// Mitsubishi GX Developer project: PLC_PCO520L2   PLC: Q06UDEH

PROGRAM MANUAL
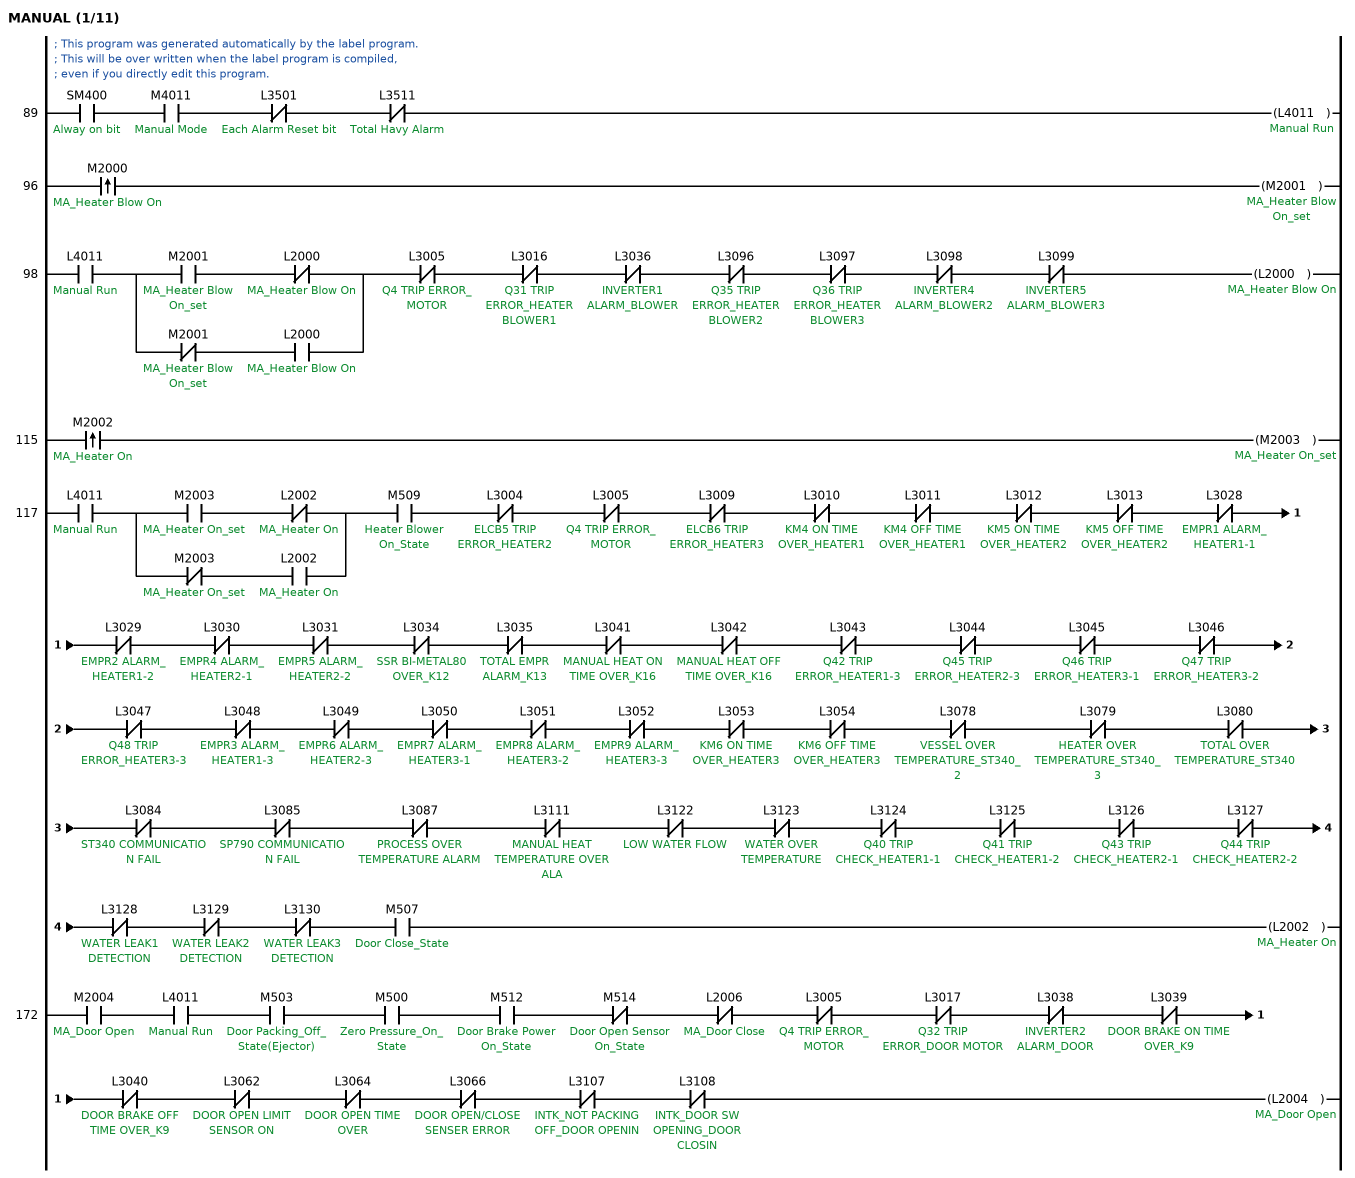
; This program was generated automatically by the label program.
; This will be over written when the label program is compiled,
; even if you directly edit this program.
89    LD      SM400  ; Alway on bit
      AND     M4011  ; Manual Mode
      ANI     L3501  ; Each Alarm Reset bit
      ANI     L3511  ; Total Havy Alarm
      OUT     L4011  ; Manual Run
; 
96    LDP     M2000  ; MA_Heater Blow On
      OUT     M2001  ; MA_Heater Blow On_set
98    LD      L4011  ; Manual Run
      LD      M2001  ; MA_Heater Blow On_set
      ANI     L2000  ; MA_Heater Blow On
      LDI     M2001  ; MA_Heater Blow On_set
      AND     L2000  ; MA_Heater Blow On
      ORB
      ANB
      ANI     L3005  ; Q4 TRIP ERROR_MOTOR
      ANI     L3016  ; Q31 TRIP ERROR_HEATER BLOWER1
      ANI     L3036  ; INVERTER1 ALARM_BLOWER
      ANI     L3096  ; Q35 TRIP ERROR_HEATER BLOWER2
      ANI     L3097  ; Q36 TRIP ERROR_HEATER BLOWER3
      ANI     L3098  ; INVERTER4 ALARM_BLOWER2
      ANI     L3099  ; INVERTER5 ALARM_BLOWER3
      OUT     L2000  ; MA_Heater Blow On
; 
115   LDP     M2002  ; MA_Heater On
      OUT     M2003  ; MA_Heater On_set
117   LD      L4011  ; Manual Run
      LD      M2003  ; MA_Heater On_set
      ANI     L2002  ; MA_Heater On
      LDI     M2003  ; MA_Heater On_set
      AND     L2002  ; MA_Heater On
      ORB
      ANB
      AND     M509  ; Heater Blower On_State
      ANI     L3004  ; ELCB5 TRIP ERROR_HEATER2
      ANI     L3005  ; Q4 TRIP ERROR_MOTOR
      ANI     L3009  ; ELCB6 TRIP ERROR_HEATER3
      ANI     L3010  ; KM4 ON TIME OVER_HEATER1
      ANI     L3011  ; KM4 OFF TIME OVER_HEATER1
      ANI     L3012  ; KM5 ON TIME OVER_HEATER2
      ANI     L3013  ; KM5 OFF TIME OVER_HEATER2
      ANI     L3028  ; EMPR1 ALARM_HEATER1-1
      ANI     L3029  ; EMPR2 ALARM_HEATER1-2
      ANI     L3030  ; EMPR4 ALARM_HEATER2-1
      ANI     L3031  ; EMPR5 ALARM_HEATER2-2
      ANI     L3034  ; SSR BI-METAL80 OVER_K12
      ANI     L3035  ; TOTAL EMPR ALARM_K13
      ANI     L3041  ; MANUAL HEAT ON TIME OVER_K16
      ANI     L3042  ; MANUAL HEAT OFF TIME OVER_K16
      ANI     L3043  ; Q42 TRIP ERROR_HEATER1-3
      ANI     L3044  ; Q45 TRIP ERROR_HEATER2-3
      ANI     L3045  ; Q46 TRIP ERROR_HEATER3-1
      ANI     L3046  ; Q47 TRIP ERROR_HEATER3-2
      ANI     L3047  ; Q48 TRIP ERROR_HEATER3-3
      ANI     L3048  ; EMPR3 ALARM_HEATER1-3
      ANI     L3049  ; EMPR6 ALARM_HEATER2-3
      ANI     L3050  ; EMPR7 ALARM_HEATER3-1
      ANI     L3051  ; EMPR8 ALARM_HEATER3-2
      ANI     L3052  ; EMPR9 ALARM_HEATER3-3
      ANI     L3053  ; KM6 ON TIME OVER_HEATER3
      ANI     L3054  ; KM6 OFF TIME OVER_HEATER3
      ANI     L3078  ; VESSEL OVER TEMPERATURE_ST340_2
      ANI     L3079  ; HEATER OVER TEMPERATURE_ST340_3
      ANI     L3080  ; TOTAL OVER TEMPERATURE_ST340
      ANI     L3084  ; ST340 COMMUNICATION FAIL
      ANI     L3085  ; SP790 COMMUNICATION FAIL
      ANI     L3087  ; PROCESS OVER TEMPERATURE ALARM
      ANI     L3111  ; MANUAL HEAT TEMPERATURE OVER ALA
      ANI     L3122  ; LOW WATER FLOW
      ANI     L3123  ; WATER OVER TEMPERATURE
      ANI     L3124  ; Q40 TRIP CHECK_HEATER1-1
      ANI     L3125  ; Q41 TRIP CHECK_HEATER1-2
      ANI     L3126  ; Q43 TRIP CHECK_HEATER2-1
      ANI     L3127  ; Q44 TRIP CHECK_HEATER2-2
      ANI     L3128  ; WATER LEAK1 DETECTION
      ANI     L3129  ; WATER LEAK2 DETECTION
      ANI     L3130  ; WATER LEAK3 DETECTION
      AND     M507  ; Door Close_State
      OUT     L2002  ; MA_Heater On
; 
172   LD      M2004  ; MA_Door Open
      AND     L4011  ; Manual Run
      AND     M503  ; Door Packing_Off_State(Ejector)
      AND     M500  ; Zero Pressure_On_State
      AND     M512  ; Door Brake Power On_State
      ANI     M514  ; Door Open Sensor On_State
      ANI     L2006  ; MA_Door Close
      ANI     L3005  ; Q4 TRIP ERROR_MOTOR
      ANI     L3017  ; Q32 TRIP ERROR_DOOR MOTOR
      ANI     L3038  ; INVERTER2 ALARM_DOOR
      ANI     L3039  ; DOOR BRAKE ON TIME OVER_K9
      ANI     L3040  ; DOOR BRAKE OFF TIME OVER_K9
      ANI     L3062  ; DOOR OPEN LIMIT SENSOR ON
      ANI     L3064  ; DOOR OPEN TIME OVER
      ANI     L3066  ; DOOR OPEN/CLOSE SENSER ERROR
      ANI     L3107  ; INTK_NOT PACKING OFF_DOOR OPENIN
      ANI     L3108  ; INTK_DOOR SW OPENING_DOOR CLOSIN
      OUT     L2004  ; MA_Door Open
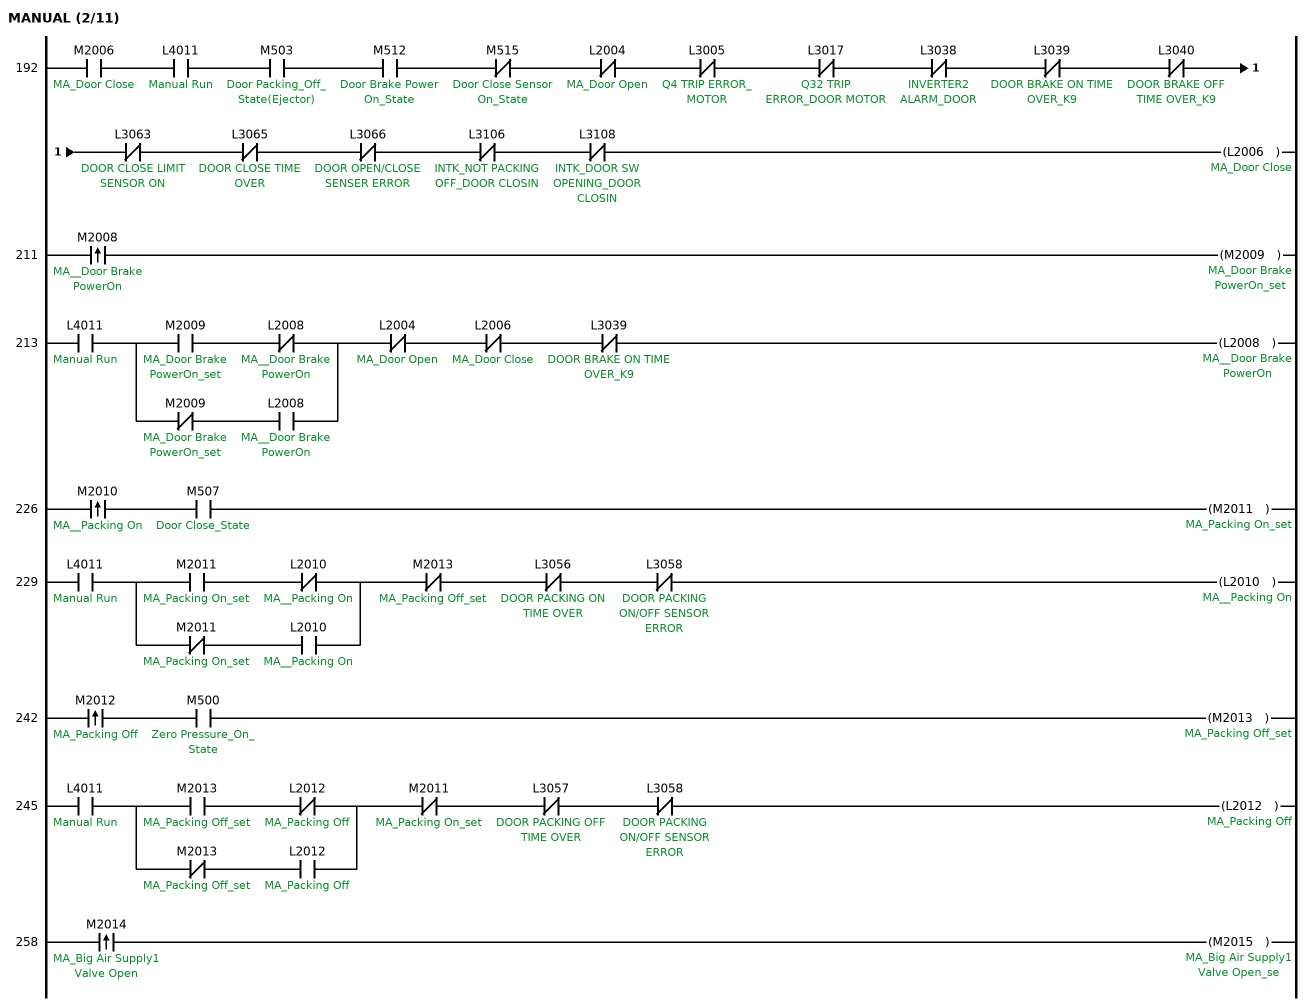
; 
192   LD      M2006  ; MA_Door Close
      AND     L4011  ; Manual Run
      AND     M503  ; Door Packing_Off_State(Ejector)
      AND     M512  ; Door Brake Power On_State
      ANI     M515  ; Door Close Sensor On_State
      ANI     L2004  ; MA_Door Open
      ANI     L3005  ; Q4 TRIP ERROR_MOTOR
      ANI     L3017  ; Q32 TRIP ERROR_DOOR MOTOR
      ANI     L3038  ; INVERTER2 ALARM_DOOR
      ANI     L3039  ; DOOR BRAKE ON TIME OVER_K9
      ANI     L3040  ; DOOR BRAKE OFF TIME OVER_K9
      ANI     L3063  ; DOOR CLOSE LIMIT SENSOR ON
      ANI     L3065  ; DOOR CLOSE TIME OVER
      ANI     L3066  ; DOOR OPEN/CLOSE SENSER ERROR
      ANI     L3106  ; INTK_NOT PACKING OFF_DOOR CLOSIN
      ANI     L3108  ; INTK_DOOR SW OPENING_DOOR CLOSIN
      OUT     L2006  ; MA_Door Close
; 
211   LDP     M2008  ; MA__Door Brake PowerOn
      OUT     M2009  ; MA_Door Brake PowerOn_set
213   LD      L4011  ; Manual Run
      LD      M2009  ; MA_Door Brake PowerOn_set
      ANI     L2008  ; MA__Door Brake PowerOn
      LDI     M2009  ; MA_Door Brake PowerOn_set
      AND     L2008  ; MA__Door Brake PowerOn
      ORB
      ANB
      ANI     L2004  ; MA_Door Open
      ANI     L2006  ; MA_Door Close
      ANI     L3039  ; DOOR BRAKE ON TIME OVER_K9
      OUT     L2008  ; MA__Door Brake PowerOn
; 
226   LDP     M2010  ; MA__Packing On
      AND     M507  ; Door Close_State
      OUT     M2011  ; MA_Packing On_set
229   LD      L4011  ; Manual Run
      LD      M2011  ; MA_Packing On_set
      ANI     L2010  ; MA__Packing On
      LDI     M2011  ; MA_Packing On_set
      AND     L2010  ; MA__Packing On
      ORB
      ANB
      ANI     M2013  ; MA_Packing Off_set
      ANI     L3056  ; DOOR PACKING ON TIME OVER
      ANI     L3058  ; DOOR PACKING ON/OFF SENSOR ERROR
      OUT     L2010  ; MA__Packing On
; 
242   LDP     M2012  ; MA_Packing Off
      AND     M500  ; Zero Pressure_On_State
      OUT     M2013  ; MA_Packing Off_set
245   LD      L4011  ; Manual Run
      LD      M2013  ; MA_Packing Off_set
      ANI     L2012  ; MA_Packing Off
      LDI     M2013  ; MA_Packing Off_set
      AND     L2012  ; MA_Packing Off
      ORB
      ANB
      ANI     M2011  ; MA_Packing On_set
      ANI     L3057  ; DOOR PACKING OFF TIME OVER
      ANI     L3058  ; DOOR PACKING ON/OFF SENSOR ERROR
      OUT     L2012  ; MA_Packing Off
; 
258   LDP     M2014  ; MA_Big Air Supply1 Valve Open
      OUT     M2015  ; MA_Big Air Supply1 Valve Open_se
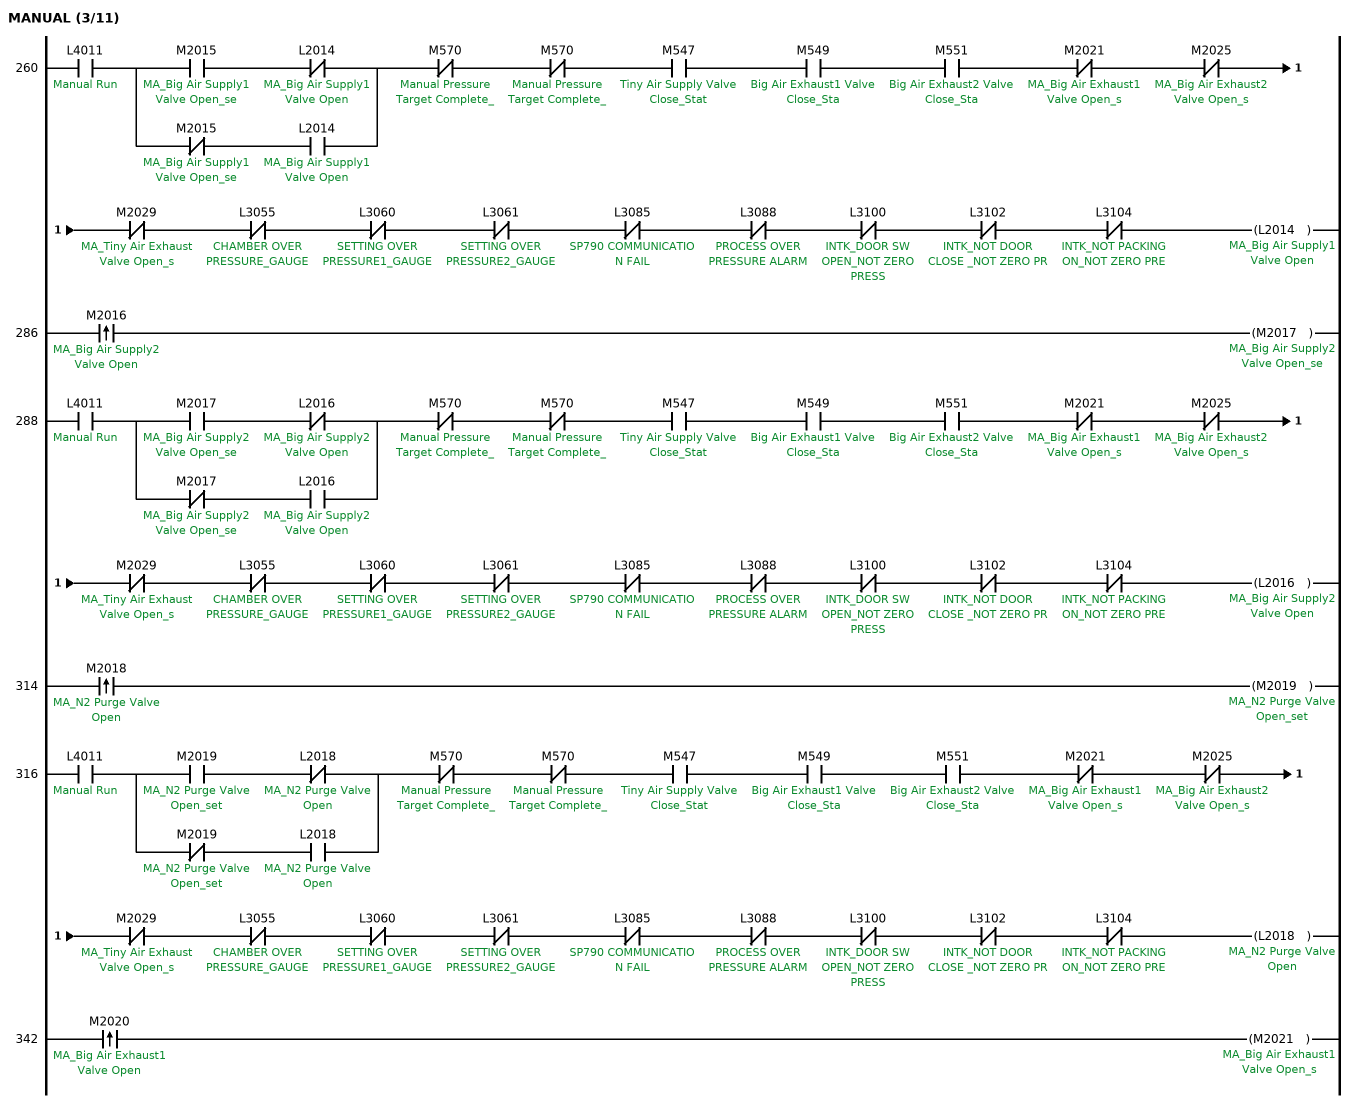
260   LD      L4011  ; Manual Run
      LD      M2015  ; MA_Big Air Supply1 Valve Open_se
      ANI     L2014  ; MA_Big Air Supply1 Valve Open
      LDI     M2015  ; MA_Big Air Supply1 Valve Open_se
      AND     L2014  ; MA_Big Air Supply1 Valve Open
      ORB
      ANB
      ANI     M570  ; Manual Pressure Target Complete_
      ANI     M570  ; Manual Pressure Target Complete_
      AND     M547  ; Tiny Air Supply Valve Close_Stat
      AND     M549  ; Big Air Exhaust1 Valve Close_Sta
      AND     M551  ; Big Air Exhaust2 Valve Close_Sta
      ANI     M2021  ; MA_Big Air Exhaust1 Valve Open_s
      ANI     M2025  ; MA_Big Air Exhaust2 Valve Open_s
      ANI     M2029  ; MA_Tiny Air Exhaust Valve Open_s
      ANI     L3055  ; CHAMBER OVER PRESSURE_GAUGE
      ANI     L3060  ; SETTING OVER PRESSURE1_GAUGE
      ANI     L3061  ; SETTING OVER PRESSURE2_GAUGE
      ANI     L3085  ; SP790 COMMUNICATION FAIL
      ANI     L3088  ; PROCESS OVER PRESSURE ALARM
      ANI     L3100  ; INTK_DOOR SW OPEN_NOT ZERO PRESS
      ANI     L3102  ; INTK_NOT DOOR CLOSE _NOT ZERO PR
      ANI     L3104  ; INTK_NOT PACKING ON_NOT ZERO PRE
      OUT     L2014  ; MA_Big Air Supply1 Valve Open
; 
286   LDP     M2016  ; MA_Big Air Supply2 Valve Open
      OUT     M2017  ; MA_Big Air Supply2 Valve Open_se
288   LD      L4011  ; Manual Run
      LD      M2017  ; MA_Big Air Supply2 Valve Open_se
      ANI     L2016  ; MA_Big Air Supply2 Valve Open
      LDI     M2017  ; MA_Big Air Supply2 Valve Open_se
      AND     L2016  ; MA_Big Air Supply2 Valve Open
      ORB
      ANB
      ANI     M570  ; Manual Pressure Target Complete_
      ANI     M570  ; Manual Pressure Target Complete_
      AND     M547  ; Tiny Air Supply Valve Close_Stat
      AND     M549  ; Big Air Exhaust1 Valve Close_Sta
      AND     M551  ; Big Air Exhaust2 Valve Close_Sta
      ANI     M2021  ; MA_Big Air Exhaust1 Valve Open_s
      ANI     M2025  ; MA_Big Air Exhaust2 Valve Open_s
      ANI     M2029  ; MA_Tiny Air Exhaust Valve Open_s
      ANI     L3055  ; CHAMBER OVER PRESSURE_GAUGE
      ANI     L3060  ; SETTING OVER PRESSURE1_GAUGE
      ANI     L3061  ; SETTING OVER PRESSURE2_GAUGE
      ANI     L3085  ; SP790 COMMUNICATION FAIL
      ANI     L3088  ; PROCESS OVER PRESSURE ALARM
      ANI     L3100  ; INTK_DOOR SW OPEN_NOT ZERO PRESS
      ANI     L3102  ; INTK_NOT DOOR CLOSE _NOT ZERO PR
      ANI     L3104  ; INTK_NOT PACKING ON_NOT ZERO PRE
      OUT     L2016  ; MA_Big Air Supply2 Valve Open
; 
314   LDP     M2018  ; MA_N2 Purge Valve Open
      OUT     M2019  ; MA_N2 Purge Valve Open_set
316   LD      L4011  ; Manual Run
      LD      M2019  ; MA_N2 Purge Valve Open_set
      ANI     L2018  ; MA_N2 Purge Valve Open
      LDI     M2019  ; MA_N2 Purge Valve Open_set
      AND     L2018  ; MA_N2 Purge Valve Open
      ORB
      ANB
      ANI     M570  ; Manual Pressure Target Complete_
      ANI     M570  ; Manual Pressure Target Complete_
      AND     M547  ; Tiny Air Supply Valve Close_Stat
      AND     M549  ; Big Air Exhaust1 Valve Close_Sta
      AND     M551  ; Big Air Exhaust2 Valve Close_Sta
      ANI     M2021  ; MA_Big Air Exhaust1 Valve Open_s
      ANI     M2025  ; MA_Big Air Exhaust2 Valve Open_s
      ANI     M2029  ; MA_Tiny Air Exhaust Valve Open_s
      ANI     L3055  ; CHAMBER OVER PRESSURE_GAUGE
      ANI     L3060  ; SETTING OVER PRESSURE1_GAUGE
      ANI     L3061  ; SETTING OVER PRESSURE2_GAUGE
      ANI     L3085  ; SP790 COMMUNICATION FAIL
      ANI     L3088  ; PROCESS OVER PRESSURE ALARM
      ANI     L3100  ; INTK_DOOR SW OPEN_NOT ZERO PRESS
      ANI     L3102  ; INTK_NOT DOOR CLOSE _NOT ZERO PR
      ANI     L3104  ; INTK_NOT PACKING ON_NOT ZERO PRE
      OUT     L2018  ; MA_N2 Purge Valve Open
; 
342   LDP     M2020  ; MA_Big Air Exhaust1 Valve Open
      OUT     M2021  ; MA_Big Air Exhaust1 Valve Open_s
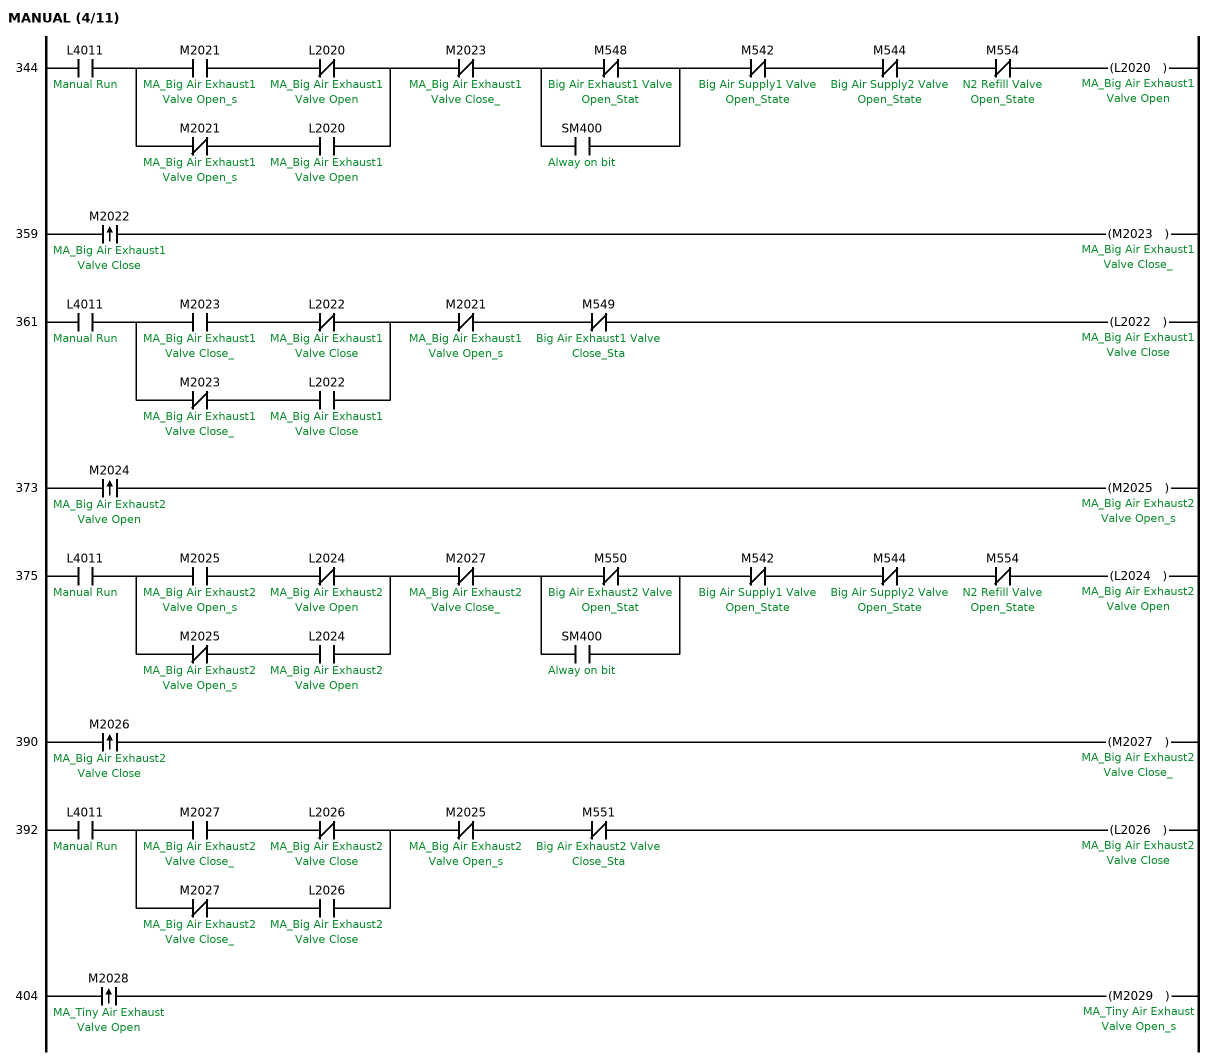
344   LD      L4011  ; Manual Run
      LD      M2021  ; MA_Big Air Exhaust1 Valve Open_s
      ANI     L2020  ; MA_Big Air Exhaust1 Valve Open
      LDI     M2021  ; MA_Big Air Exhaust1 Valve Open_s
      AND     L2020  ; MA_Big Air Exhaust1 Valve Open
      ORB
      ANB
      ANI     M2023  ; MA_Big Air Exhaust1 Valve Close_
      LDI     M548  ; Big Air Exhaust1 Valve Open_Stat
      OR      SM400  ; Alway on bit
      ANB
      ANI     M542  ; Big Air Supply1 Valve Open_State
      ANI     M544  ; Big Air Supply2 Valve Open_State
      ANI     M554  ; N2 Refill Valve Open_State
      OUT     L2020  ; MA_Big Air Exhaust1 Valve Open
359   LDP     M2022  ; MA_Big Air Exhaust1 Valve Close
      OUT     M2023  ; MA_Big Air Exhaust1 Valve Close_
361   LD      L4011  ; Manual Run
      LD      M2023  ; MA_Big Air Exhaust1 Valve Close_
      ANI     L2022  ; MA_Big Air Exhaust1 Valve Close
      LDI     M2023  ; MA_Big Air Exhaust1 Valve Close_
      AND     L2022  ; MA_Big Air Exhaust1 Valve Close
      ORB
      ANB
      ANI     M2021  ; MA_Big Air Exhaust1 Valve Open_s
      ANI     M549  ; Big Air Exhaust1 Valve Close_Sta
      OUT     L2022  ; MA_Big Air Exhaust1 Valve Close
; 
373   LDP     M2024  ; MA_Big Air Exhaust2 Valve Open
      OUT     M2025  ; MA_Big Air Exhaust2 Valve Open_s
375   LD      L4011  ; Manual Run
      LD      M2025  ; MA_Big Air Exhaust2 Valve Open_s
      ANI     L2024  ; MA_Big Air Exhaust2 Valve Open
      LDI     M2025  ; MA_Big Air Exhaust2 Valve Open_s
      AND     L2024  ; MA_Big Air Exhaust2 Valve Open
      ORB
      ANB
      ANI     M2027  ; MA_Big Air Exhaust2 Valve Close_
      LDI     M550  ; Big Air Exhaust2 Valve Open_Stat
      OR      SM400  ; Alway on bit
      ANB
      ANI     M542  ; Big Air Supply1 Valve Open_State
      ANI     M544  ; Big Air Supply2 Valve Open_State
      ANI     M554  ; N2 Refill Valve Open_State
      OUT     L2024  ; MA_Big Air Exhaust2 Valve Open
390   LDP     M2026  ; MA_Big Air Exhaust2 Valve Close
      OUT     M2027  ; MA_Big Air Exhaust2 Valve Close_
392   LD      L4011  ; Manual Run
      LD      M2027  ; MA_Big Air Exhaust2 Valve Close_
      ANI     L2026  ; MA_Big Air Exhaust2 Valve Close
      LDI     M2027  ; MA_Big Air Exhaust2 Valve Close_
      AND     L2026  ; MA_Big Air Exhaust2 Valve Close
      ORB
      ANB
      ANI     M2025  ; MA_Big Air Exhaust2 Valve Open_s
      ANI     M551  ; Big Air Exhaust2 Valve Close_Sta
      OUT     L2026  ; MA_Big Air Exhaust2 Valve Close
; 
404   LDP     M2028  ; MA_Tiny Air Exhaust Valve Open
      OUT     M2029  ; MA_Tiny Air Exhaust Valve Open_s
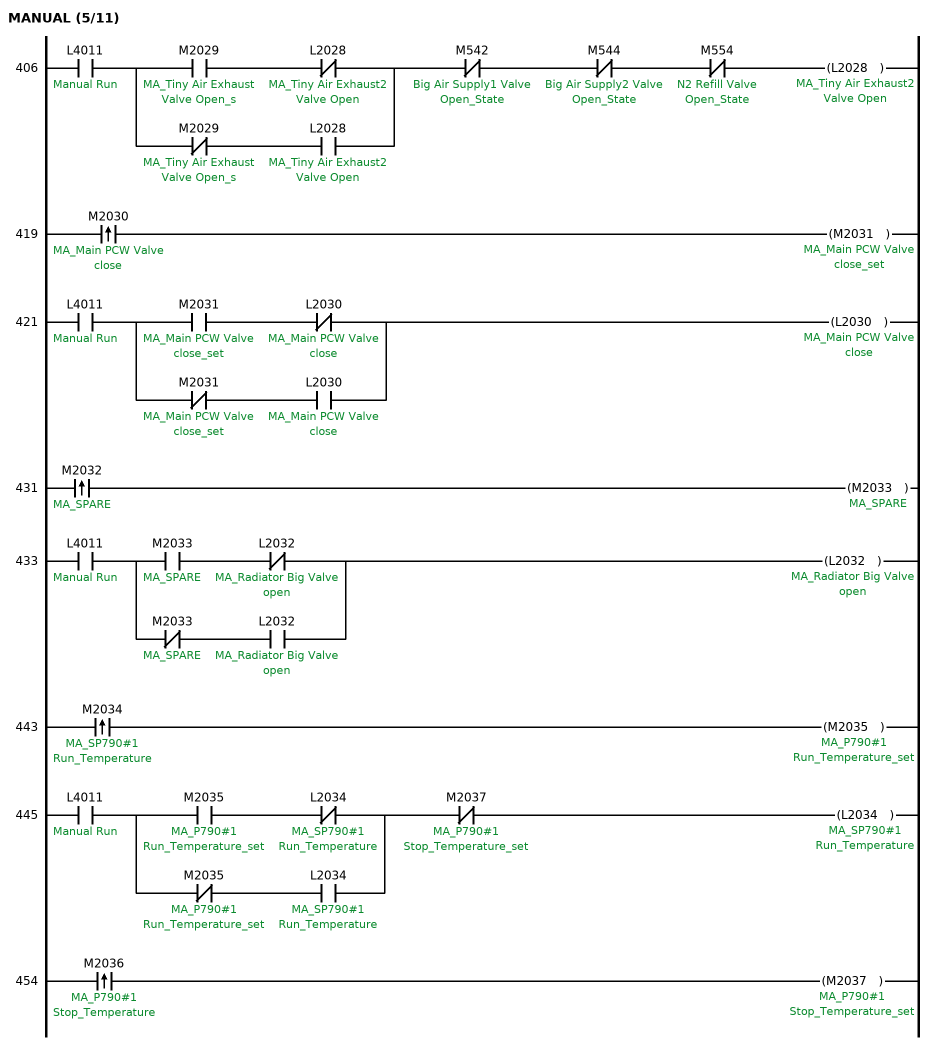
406   LD      L4011  ; Manual Run
      LD      M2029  ; MA_Tiny Air Exhaust Valve Open_s
      ANI     L2028  ; MA_Tiny Air Exhaust2 Valve Open
      LDI     M2029  ; MA_Tiny Air Exhaust Valve Open_s
      AND     L2028  ; MA_Tiny Air Exhaust2 Valve Open
      ORB
      ANB
      ANI     M542  ; Big Air Supply1 Valve Open_State
      ANI     M544  ; Big Air Supply2 Valve Open_State
      ANI     M554  ; N2 Refill Valve Open_State
      OUT     L2028  ; MA_Tiny Air Exhaust2 Valve Open
; 
419   LDP     M2030  ; MA_Main PCW Valve close
      OUT     M2031  ; MA_Main PCW Valve close_set
421   LD      L4011  ; Manual Run
      LD      M2031  ; MA_Main PCW Valve close_set
      ANI     L2030  ; MA_Main PCW Valve close
      LDI     M2031  ; MA_Main PCW Valve close_set
      AND     L2030  ; MA_Main PCW Valve close
      ORB
      ANB
      OUT     L2030  ; MA_Main PCW Valve close
; 
431   LDP     M2032  ; MA_SPARE
      OUT     M2033  ; MA_SPARE
433   LD      L4011  ; Manual Run
      LD      M2033  ; MA_SPARE
      ANI     L2032  ; MA_Radiator Big Valve open
      LDI     M2033  ; MA_SPARE
      AND     L2032  ; MA_Radiator Big Valve open
      ORB
      ANB
      OUT     L2032  ; MA_Radiator Big Valve open
; 
443   LDP     M2034  ; MA_SP790#1 Run_Temperature
      OUT     M2035  ; MA_P790#1 Run_Temperature_set
445   LD      L4011  ; Manual Run
      LD      M2035  ; MA_P790#1 Run_Temperature_set
      ANI     L2034  ; MA_SP790#1 Run_Temperature
      LDI     M2035  ; MA_P790#1 Run_Temperature_set
      AND     L2034  ; MA_SP790#1 Run_Temperature
      ORB
      ANB
      ANI     M2037  ; MA_P790#1 Stop_Temperature_set
      OUT     L2034  ; MA_SP790#1 Run_Temperature
454   LDP     M2036  ; MA_P790#1 Stop_Temperature
      OUT     M2037  ; MA_P790#1 Stop_Temperature_set
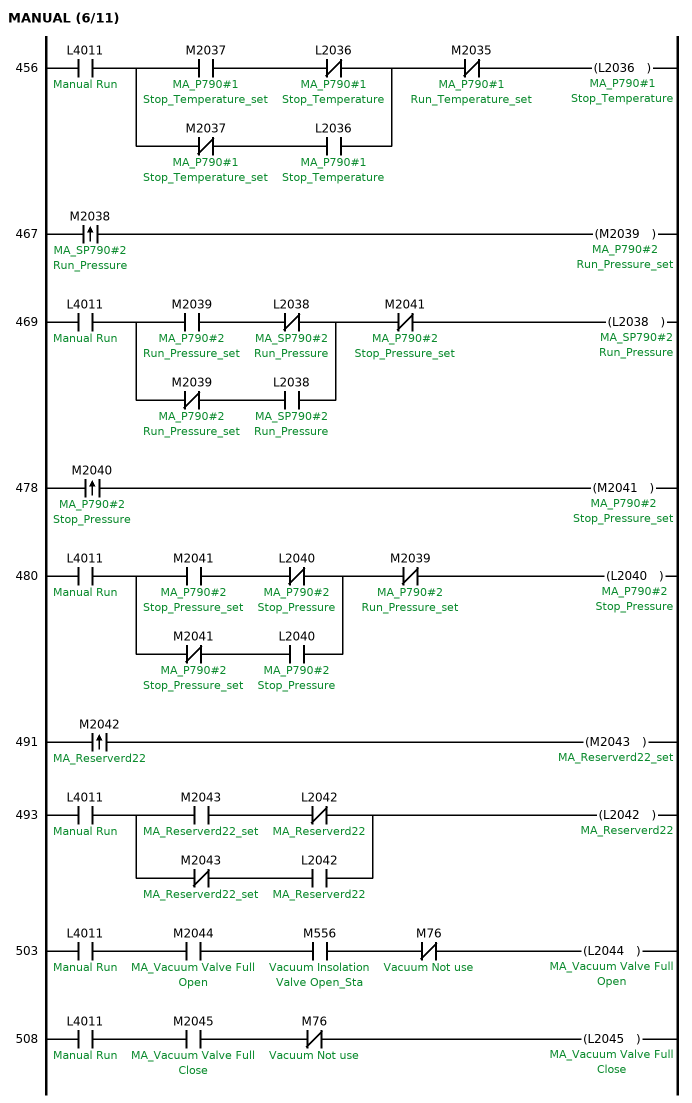
456   LD      L4011  ; Manual Run
      LD      M2037  ; MA_P790#1 Stop_Temperature_set
      ANI     L2036  ; MA_P790#1 Stop_Temperature
      LDI     M2037  ; MA_P790#1 Stop_Temperature_set
      AND     L2036  ; MA_P790#1 Stop_Temperature
      ORB
      ANB
      ANI     M2035  ; MA_P790#1 Run_Temperature_set
      OUT     L2036  ; MA_P790#1 Stop_Temperature
; 
467   LDP     M2038  ; MA_SP790#2 Run_Pressure
      OUT     M2039  ; MA_P790#2 Run_Pressure_set
469   LD      L4011  ; Manual Run
      LD      M2039  ; MA_P790#2 Run_Pressure_set
      ANI     L2038  ; MA_SP790#2 Run_Pressure
      LDI     M2039  ; MA_P790#2 Run_Pressure_set
      AND     L2038  ; MA_SP790#2 Run_Pressure
      ORB
      ANB
      ANI     M2041  ; MA_P790#2 Stop_Pressure_set
      OUT     L2038  ; MA_SP790#2 Run_Pressure
478   LDP     M2040  ; MA_P790#2 Stop_Pressure
      OUT     M2041  ; MA_P790#2 Stop_Pressure_set
480   LD      L4011  ; Manual Run
      LD      M2041  ; MA_P790#2 Stop_Pressure_set
      ANI     L2040  ; MA_P790#2 Stop_Pressure
      LDI     M2041  ; MA_P790#2 Stop_Pressure_set
      AND     L2040  ; MA_P790#2 Stop_Pressure
      ORB
      ANB
      ANI     M2039  ; MA_P790#2 Run_Pressure_set
      OUT     L2040  ; MA_P790#2 Stop_Pressure
; 
491   LDP     M2042  ; MA_Reserverd22
      OUT     M2043  ; MA_Reserverd22_set
493   LD      L4011  ; Manual Run
      LD      M2043  ; MA_Reserverd22_set
      ANI     L2042  ; MA_Reserverd22
      LDI     M2043  ; MA_Reserverd22_set
      AND     L2042  ; MA_Reserverd22
      ORB
      ANB
      OUT     L2042  ; MA_Reserverd22
; 
503   LD      L4011  ; Manual Run
      AND     M2044  ; MA_Vacuum Valve Full Open
      AND     M556  ; Vacuum Insolation Valve Open_Sta
      ANI     M76  ; Vacuum Not use
      OUT     L2044  ; MA_Vacuum Valve Full Open
508   LD      L4011  ; Manual Run
      AND     M2045  ; MA_Vacuum Valve Full Close
      ANI     M76  ; Vacuum Not use
      OUT     L2045  ; MA_Vacuum Valve Full Close
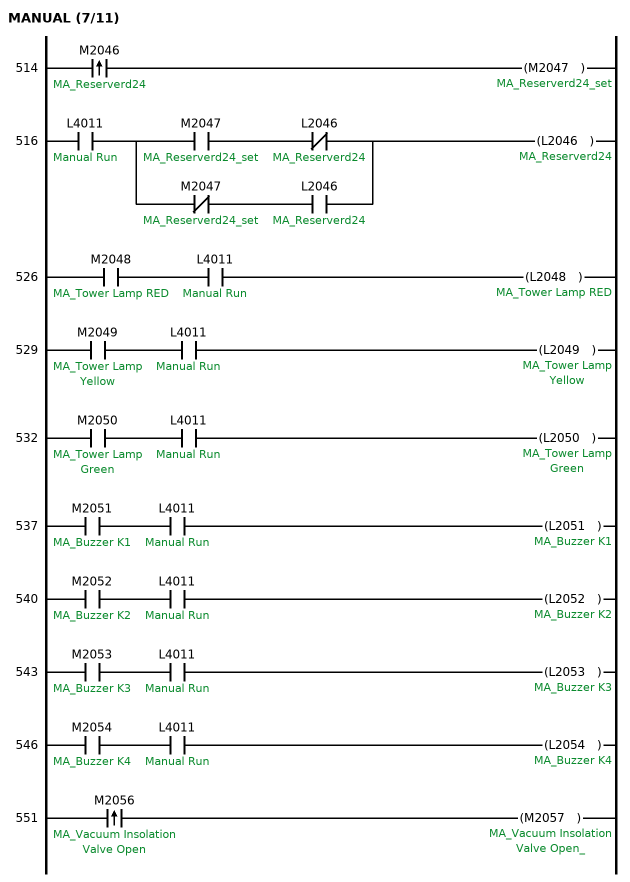
; 
514   LDP     M2046  ; MA_Reserverd24
      OUT     M2047  ; MA_Reserverd24_set
516   LD      L4011  ; Manual Run
      LD      M2047  ; MA_Reserverd24_set
      ANI     L2046  ; MA_Reserverd24
      LDI     M2047  ; MA_Reserverd24_set
      AND     L2046  ; MA_Reserverd24
      ORB
      ANB
      OUT     L2046  ; MA_Reserverd24
; 
526   LD      M2048  ; MA_Tower Lamp RED
      AND     L4011  ; Manual Run
      OUT     L2048  ; MA_Tower Lamp RED
529   LD      M2049  ; MA_Tower Lamp Yellow
      AND     L4011  ; Manual Run
      OUT     L2049  ; MA_Tower Lamp Yellow
532   LD      M2050  ; MA_Tower Lamp Green
      AND     L4011  ; Manual Run
      OUT     L2050  ; MA_Tower Lamp Green
; 
537   LD      M2051  ; MA_Buzzer K1
      AND     L4011  ; Manual Run
      OUT     L2051  ; MA_Buzzer K1
540   LD      M2052  ; MA_Buzzer K2
      AND     L4011  ; Manual Run
      OUT     L2052  ; MA_Buzzer K2
543   LD      M2053  ; MA_Buzzer K3
      AND     L4011  ; Manual Run
      OUT     L2053  ; MA_Buzzer K3
546   LD      M2054  ; MA_Buzzer K4
      AND     L4011  ; Manual Run
      OUT     L2054  ; MA_Buzzer K4
; 
551   LDP     M2056  ; MA_Vacuum Insolation Valve Open
      OUT     M2057  ; MA_Vacuum Insolation Valve Open_
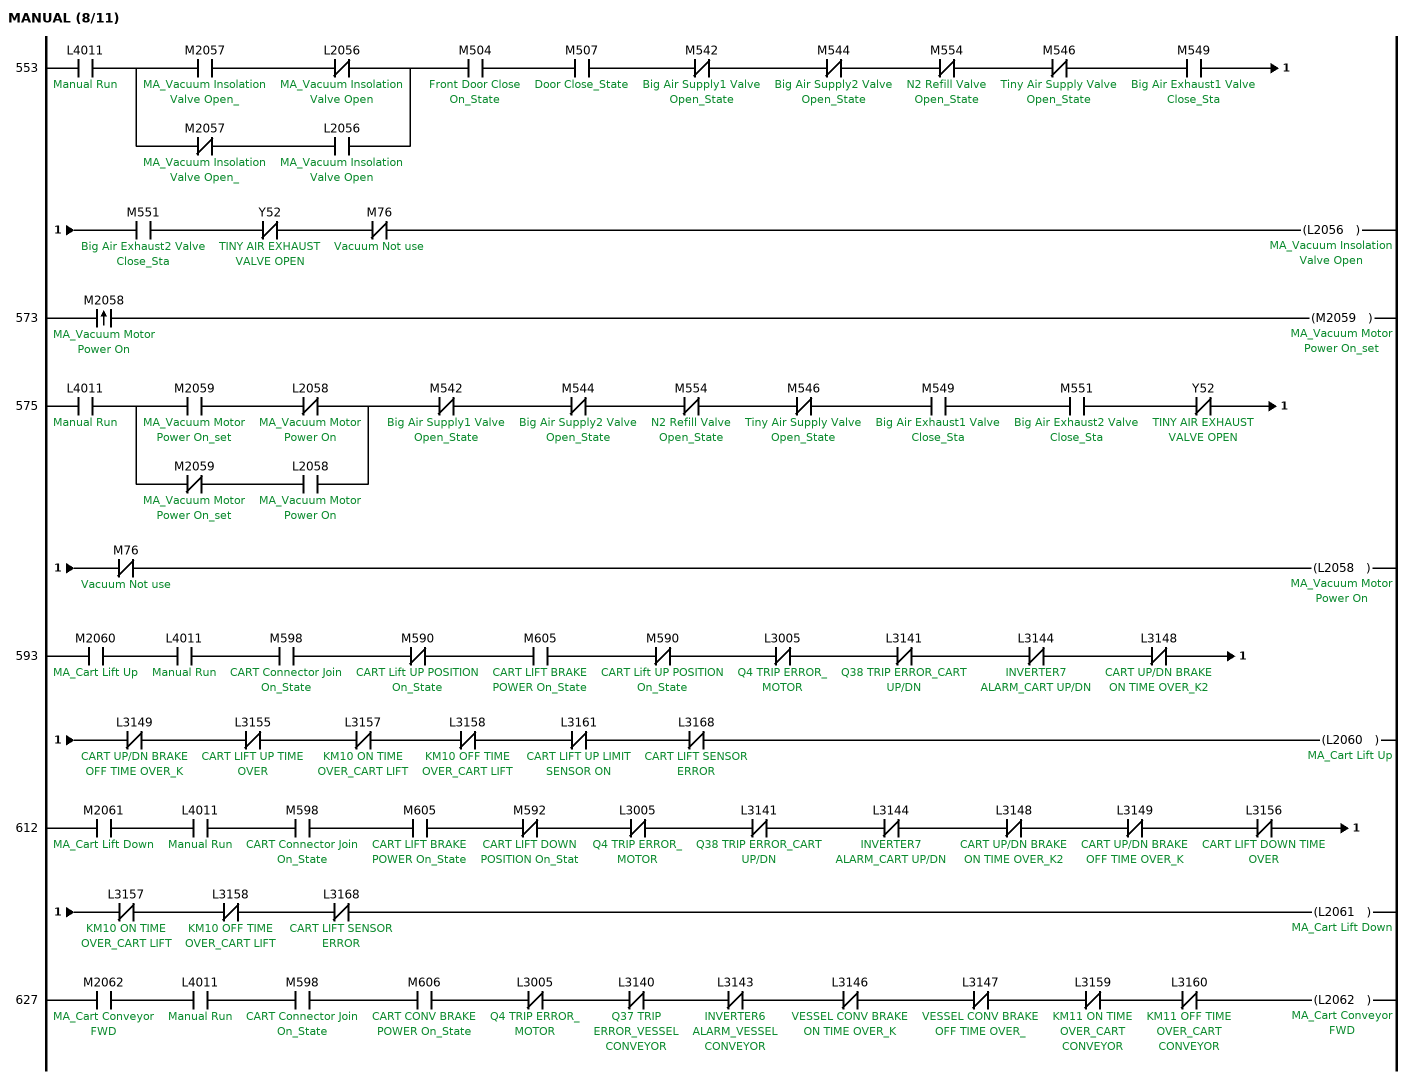
553   LD      L4011  ; Manual Run
      LD      M2057  ; MA_Vacuum Insolation Valve Open_
      ANI     L2056  ; MA_Vacuum Insolation Valve Open
      LDI     M2057  ; MA_Vacuum Insolation Valve Open_
      AND     L2056  ; MA_Vacuum Insolation Valve Open
      ORB
      ANB
      AND     M504  ; Front Door Close On_State
      AND     M507  ; Door Close_State
      ANI     M542  ; Big Air Supply1 Valve Open_State
      ANI     M544  ; Big Air Supply2 Valve Open_State
      ANI     M554  ; N2 Refill Valve Open_State
      ANI     M546  ; Tiny Air Supply Valve Open_State
      AND     M549  ; Big Air Exhaust1 Valve Close_Sta
      AND     M551  ; Big Air Exhaust2 Valve Close_Sta
      ANI     Y52  ; TINY AIR EXHAUST VALVE OPEN
      ANI     M76  ; Vacuum Not use
      OUT     L2056  ; MA_Vacuum Insolation Valve Open
; 
573   LDP     M2058  ; MA_Vacuum Motor Power On
      OUT     M2059  ; MA_Vacuum Motor Power On_set
575   LD      L4011  ; Manual Run
      LD      M2059  ; MA_Vacuum Motor Power On_set
      ANI     L2058  ; MA_Vacuum Motor Power On
      LDI     M2059  ; MA_Vacuum Motor Power On_set
      AND     L2058  ; MA_Vacuum Motor Power On
      ORB
      ANB
      ANI     M542  ; Big Air Supply1 Valve Open_State
      ANI     M544  ; Big Air Supply2 Valve Open_State
      ANI     M554  ; N2 Refill Valve Open_State
      ANI     M546  ; Tiny Air Supply Valve Open_State
      AND     M549  ; Big Air Exhaust1 Valve Close_Sta
      AND     M551  ; Big Air Exhaust2 Valve Close_Sta
      ANI     Y52  ; TINY AIR EXHAUST VALVE OPEN
      ANI     M76  ; Vacuum Not use
      OUT     L2058  ; MA_Vacuum Motor Power On
; 
593   LD      M2060  ; MA_Cart Lift Up
      AND     L4011  ; Manual Run
      AND     M598  ; CART Connector Join On_State
      ANI     M590  ; CART Lift UP POSITION On_State
      AND     M605  ; CART LIFT BRAKE POWER On_State
      ANI     M590  ; CART Lift UP POSITION On_State
      ANI     L3005  ; Q4 TRIP ERROR_MOTOR
      ANI     L3141  ; Q38 TRIP ERROR_CART UP/DN
      ANI     L3144  ; INVERTER7 ALARM_CART UP/DN
      ANI     L3148  ; CART UP/DN BRAKE ON TIME OVER_K2
      ANI     L3149  ; CART UP/DN BRAKE OFF TIME OVER_K
      ANI     L3155  ; CART LIFT UP TIME OVER
      ANI     L3157  ; KM10 ON TIME OVER_CART LIFT
      ANI     L3158  ; KM10 OFF TIME OVER_CART LIFT
      ANI     L3161  ; CART LIFT UP LIMIT SENSOR ON
      ANI     L3168  ; CART LIFT SENSOR ERROR
      OUT     L2060  ; MA_Cart Lift Up
; 
612   LD      M2061  ; MA_Cart Lift Down
      AND     L4011  ; Manual Run
      AND     M598  ; CART Connector Join On_State
      AND     M605  ; CART LIFT BRAKE POWER On_State
      ANI     M592  ; CART LIFT DOWN  POSITION On_Stat
      ANI     L3005  ; Q4 TRIP ERROR_MOTOR
      ANI     L3141  ; Q38 TRIP ERROR_CART UP/DN
      ANI     L3144  ; INVERTER7 ALARM_CART UP/DN
      ANI     L3148  ; CART UP/DN BRAKE ON TIME OVER_K2
      ANI     L3149  ; CART UP/DN BRAKE OFF TIME OVER_K
      ANI     L3156  ; CART LIFT DOWN TIME OVER
      ANI     L3157  ; KM10 ON TIME OVER_CART LIFT
      ANI     L3158  ; KM10 OFF TIME OVER_CART LIFT
      ANI     L3168  ; CART LIFT SENSOR ERROR
      OUT     L2061  ; MA_Cart Lift Down
627   LD      M2062  ; MA_Cart Conveyor FWD
      AND     L4011  ; Manual Run
      AND     M598  ; CART Connector Join On_State
      AND     M606  ; CART CONV BRAKE POWER On_State
      ANI     L3005  ; Q4 TRIP ERROR_MOTOR
      ANI     L3140  ; Q37 TRIP ERROR_VESSEL CONVEYOR
      ANI     L3143  ; INVERTER6 ALARM_VESSEL CONVEYOR
      ANI     L3146  ; VESSEL CONV BRAKE ON TIME OVER_K
      ANI     L3147  ; VESSEL CONV BRAKE OFF TIME OVER_
      ANI     L3159  ; KM11 ON TIME OVER_CART CONVEYOR
      ANI     L3160  ; KM11 OFF TIME OVER_CART CONVEYOR
      OUT     L2062  ; MA_Cart Conveyor FWD
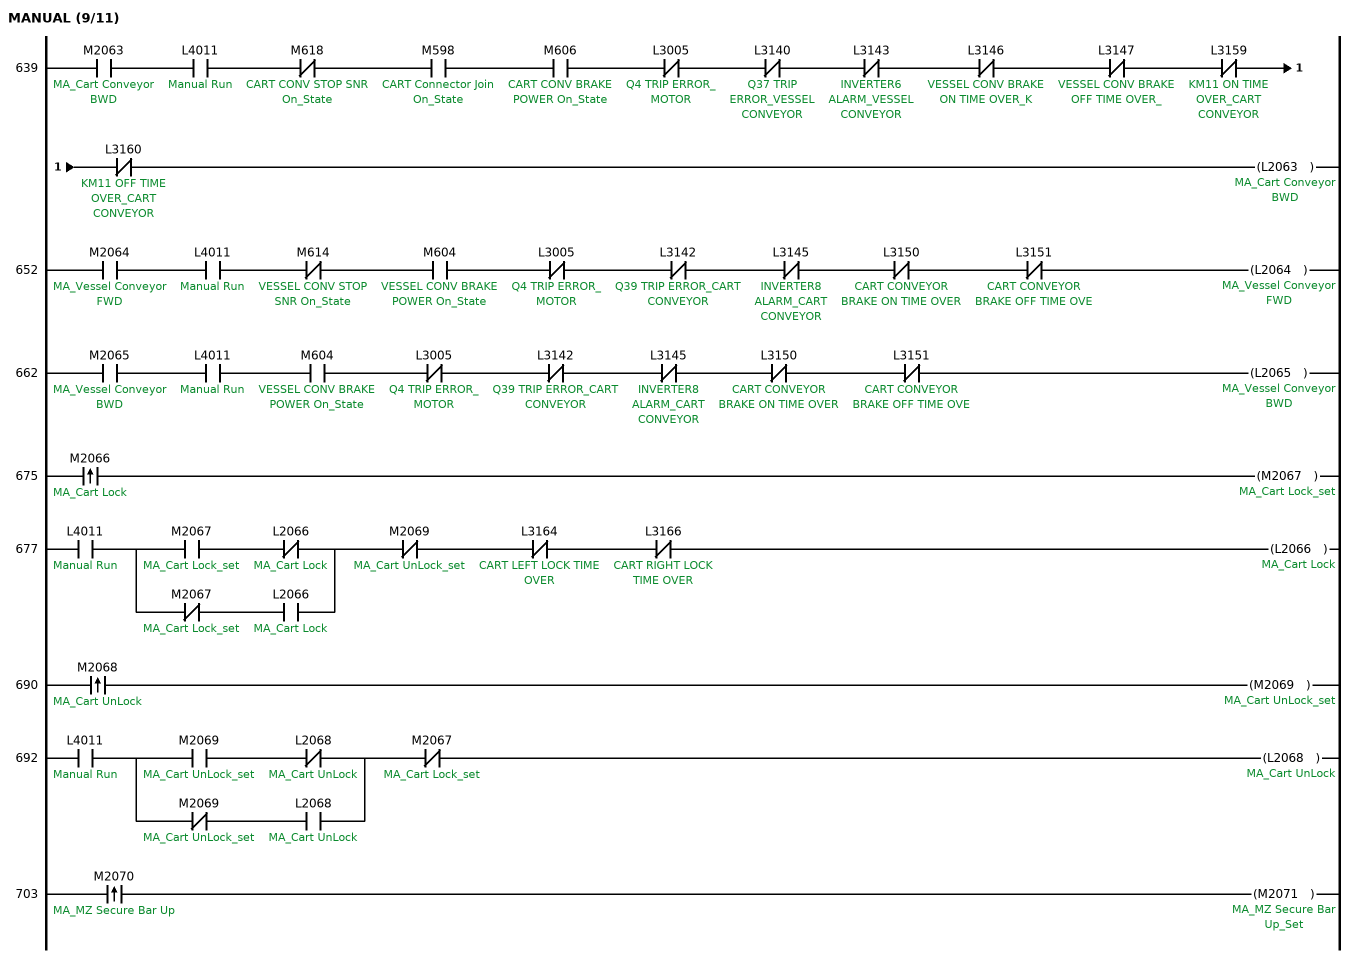
639   LD      M2063  ; MA_Cart Conveyor BWD
      AND     L4011  ; Manual Run
      ANI     M618  ; CART CONV STOP SNR On_State
      AND     M598  ; CART Connector Join On_State
      AND     M606  ; CART CONV BRAKE POWER On_State
      ANI     L3005  ; Q4 TRIP ERROR_MOTOR
      ANI     L3140  ; Q37 TRIP ERROR_VESSEL CONVEYOR
      ANI     L3143  ; INVERTER6 ALARM_VESSEL CONVEYOR
      ANI     L3146  ; VESSEL CONV BRAKE ON TIME OVER_K
      ANI     L3147  ; VESSEL CONV BRAKE OFF TIME OVER_
      ANI     L3159  ; KM11 ON TIME OVER_CART CONVEYOR
      ANI     L3160  ; KM11 OFF TIME OVER_CART CONVEYOR
      OUT     L2063  ; MA_Cart Conveyor BWD
652   LD      M2064  ; MA_Vessel Conveyor FWD
      AND     L4011  ; Manual Run
      ANI     M614  ; VESSEL CONV STOP SNR On_State
      AND     M604  ; VESSEL CONV BRAKE POWER On_State
      ANI     L3005  ; Q4 TRIP ERROR_MOTOR
      ANI     L3142  ; Q39 TRIP ERROR_CART CONVEYOR
      ANI     L3145  ; INVERTER8 ALARM_CART CONVEYOR
      ANI     L3150  ; CART CONVEYOR BRAKE ON TIME OVER
      ANI     L3151  ; CART CONVEYOR BRAKE OFF TIME OVE
      OUT     L2064  ; MA_Vessel Conveyor FWD
662   LD      M2065  ; MA_Vessel Conveyor BWD
      AND     L4011  ; Manual Run
      AND     M604  ; VESSEL CONV BRAKE POWER On_State
      ANI     L3005  ; Q4 TRIP ERROR_MOTOR
      ANI     L3142  ; Q39 TRIP ERROR_CART CONVEYOR
      ANI     L3145  ; INVERTER8 ALARM_CART CONVEYOR
      ANI     L3150  ; CART CONVEYOR BRAKE ON TIME OVER
      ANI     L3151  ; CART CONVEYOR BRAKE OFF TIME OVE
      OUT     L2065  ; MA_Vessel Conveyor BWD
; 
; 
675   LDP     M2066  ; MA_Cart Lock
      OUT     M2067  ; MA_Cart Lock_set
677   LD      L4011  ; Manual Run
      LD      M2067  ; MA_Cart Lock_set
      ANI     L2066  ; MA_Cart Lock
      LDI     M2067  ; MA_Cart Lock_set
      AND     L2066  ; MA_Cart Lock
      ORB
      ANB
      ANI     M2069  ; MA_Cart UnLock_set
      ANI     L3164  ; CART LEFT LOCK TIME OVER
      ANI     L3166  ; CART RIGHT LOCK TIME OVER
      OUT     L2066  ; MA_Cart Lock
; 
690   LDP     M2068  ; MA_Cart UnLock
      OUT     M2069  ; MA_Cart UnLock_set
692   LD      L4011  ; Manual Run
      LD      M2069  ; MA_Cart UnLock_set
      ANI     L2068  ; MA_Cart UnLock
      LDI     M2069  ; MA_Cart UnLock_set
      AND     L2068  ; MA_Cart UnLock
      ORB
      ANB
      ANI     M2067  ; MA_Cart Lock_set
      OUT     L2068  ; MA_Cart UnLock
; 
703   LDP     M2070  ; MA_MZ Secure Bar Up
      OUT     M2071  ; MA_MZ Secure Bar Up_Set
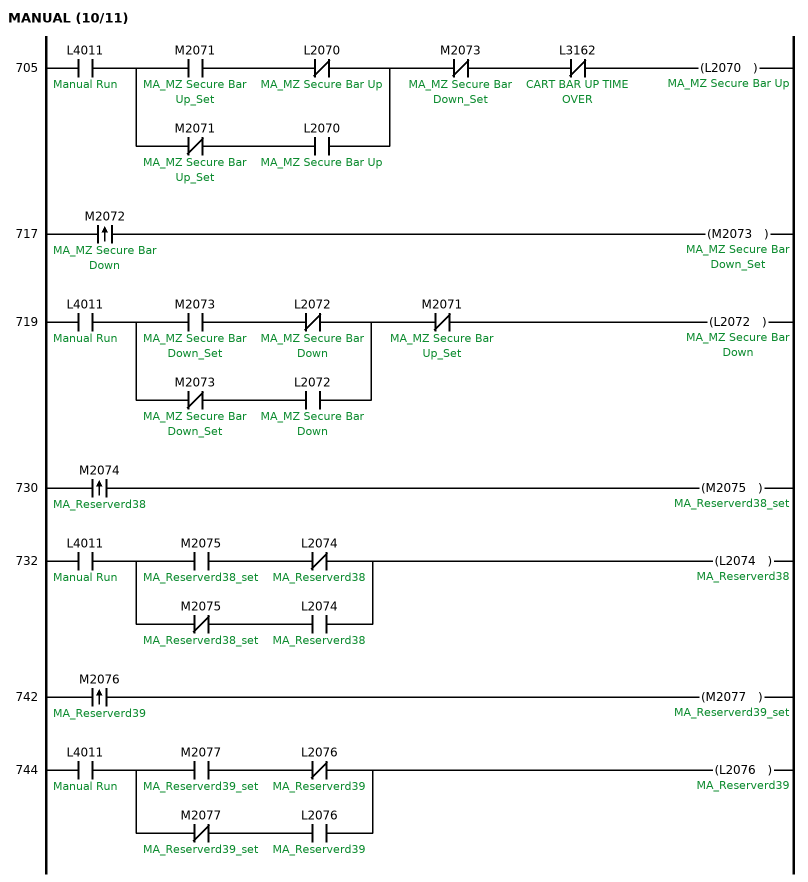
705   LD      L4011  ; Manual Run
      LD      M2071  ; MA_MZ Secure Bar Up_Set
      ANI     L2070  ; MA_MZ Secure Bar Up
      LDI     M2071  ; MA_MZ Secure Bar Up_Set
      AND     L2070  ; MA_MZ Secure Bar Up
      ORB
      ANB
      ANI     M2073  ; MA_MZ Secure Bar Down_Set
      ANI     L3162  ; CART BAR UP TIME OVER
      OUT     L2070  ; MA_MZ Secure Bar Up
; 
717   LDP     M2072  ; MA_MZ Secure Bar Down
      OUT     M2073  ; MA_MZ Secure Bar Down_Set
719   LD      L4011  ; Manual Run
      LD      M2073  ; MA_MZ Secure Bar Down_Set
      ANI     L2072  ; MA_MZ Secure Bar Down
      LDI     M2073  ; MA_MZ Secure Bar Down_Set
      AND     L2072  ; MA_MZ Secure Bar Down
      ORB
      ANB
      ANI     M2071  ; MA_MZ Secure Bar Up_Set
      OUT     L2072  ; MA_MZ Secure Bar Down
; 
730   LDP     M2074  ; MA_Reserverd38
      OUT     M2075  ; MA_Reserverd38_set
732   LD      L4011  ; Manual Run
      LD      M2075  ; MA_Reserverd38_set
      ANI     L2074  ; MA_Reserverd38
      LDI     M2075  ; MA_Reserverd38_set
      AND     L2074  ; MA_Reserverd38
      ORB
      ANB
      OUT     L2074  ; MA_Reserverd38
; 
742   LDP     M2076  ; MA_Reserverd39
      OUT     M2077  ; MA_Reserverd39_set
744   LD      L4011  ; Manual Run
      LD      M2077  ; MA_Reserverd39_set
      ANI     L2076  ; MA_Reserverd39
      LDI     M2077  ; MA_Reserverd39_set
      AND     L2076  ; MA_Reserverd39
      ORB
      ANB
      OUT     L2076  ; MA_Reserverd39
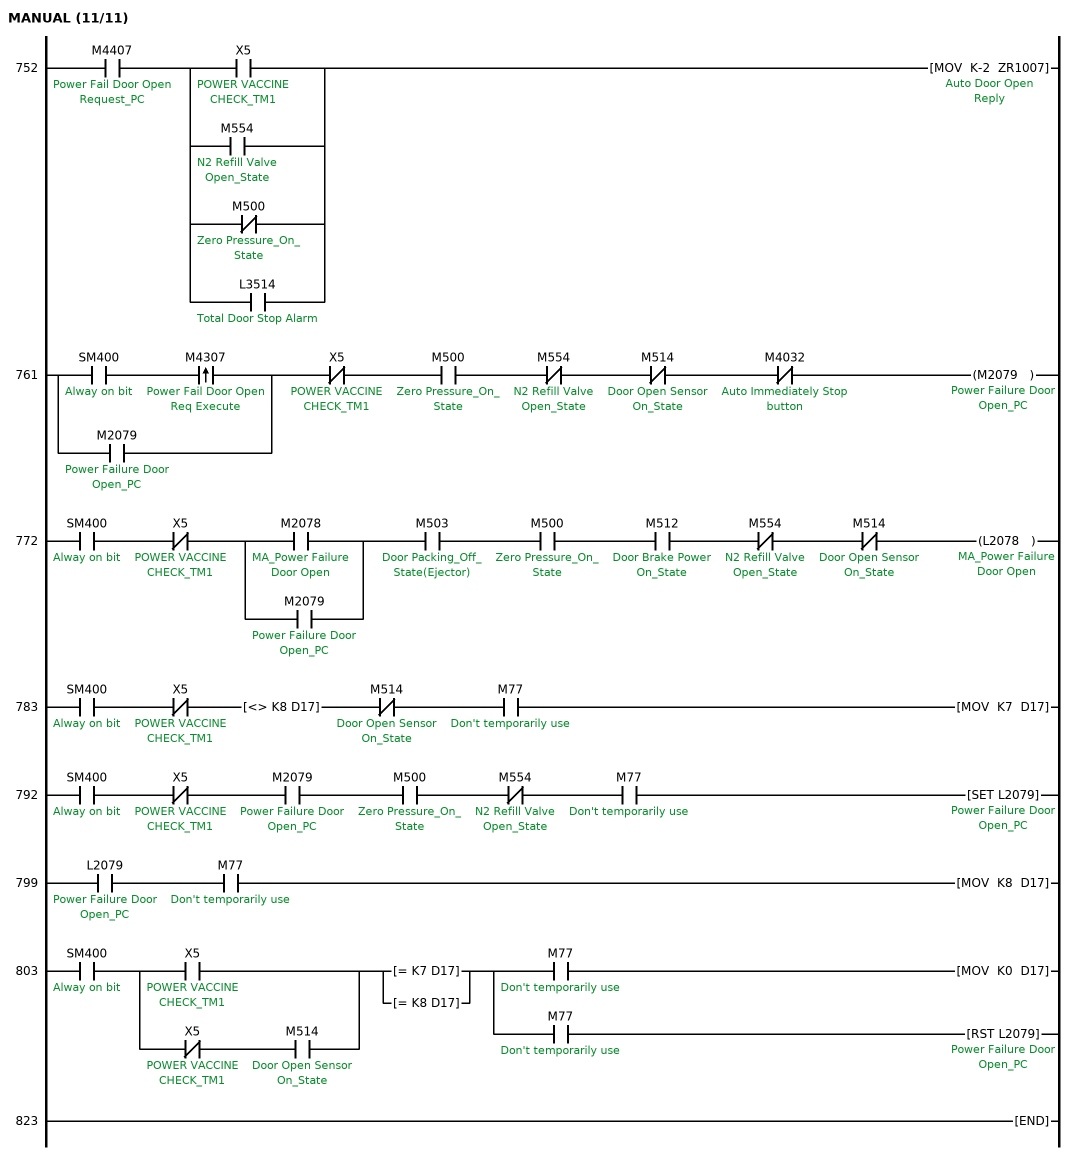
752   LD      M4407  ; Power Fail Door Open Request_PC
      LD      X5  ; POWER VACCINE CHECK_TM1
      OR      M554  ; N2 Refill Valve Open_State
      ORI     M500  ; Zero Pressure_On_State
      OR      L3514  ; Total Door Stop Alarm
      ANB
      MOV     K-2 ZR1007  ; Auto Door Open Reply
761   LD      SM400  ; Alway on bit
      ANDP    M4307  ; Power Fail Door Open Req Execute
      OR      M2079  ; Power Failure Door Open_PC
      ANI     X5  ; POWER VACCINE CHECK_TM1
      AND     M500  ; Zero Pressure_On_State
      ANI     M554  ; N2 Refill Valve Open_State
      ANI     M514  ; Door Open Sensor On_State
      ANI     M4032  ; Auto Immediately Stop button
      OUT     M2079  ; Power Failure Door Open_PC
; 
772   LD      SM400  ; Alway on bit
      ANI     X5  ; POWER VACCINE CHECK_TM1
      LD      M2078  ; MA_Power Failure Door Open
      OR      M2079  ; Power Failure Door Open_PC
      ANB
      AND     M503  ; Door Packing_Off_State(Ejector)
      AND     M500  ; Zero Pressure_On_State
      AND     M512  ; Door Brake Power On_State
      ANI     M554  ; N2 Refill Valve Open_State
      ANI     M514  ; Door Open Sensor On_State
      OUT     L2078  ; MA_Power Failure Door Open
783   LD      SM400  ; Alway on bit
      ANI     X5  ; POWER VACCINE CHECK_TM1
      AND<>   K8 D17
      ANI     M514  ; Door Open Sensor On_State
      AND     M77  ; Don't temporarily use
      MOV     K7 D17
792   LD      SM400  ; Alway on bit
      ANI     X5  ; POWER VACCINE CHECK_TM1
      AND     M2079  ; Power Failure Door Open_PC
      AND     M500  ; Zero Pressure_On_State
      ANI     M554  ; N2 Refill Valve Open_State
      AND     M77  ; Don't temporarily use
      SET     L2079  ; Power Failure Door Open_PC
799   LD      L2079  ; Power Failure Door Open_PC
      AND     M77  ; Don't temporarily use
      MOV     K8 D17
803   LD      SM400  ; Alway on bit
      LD      X5  ; POWER VACCINE CHECK_TM1
      LDI     X5  ; POWER VACCINE CHECK_TM1
      AND     M514  ; Door Open Sensor On_State
      ORB
      ANB
      LD=     K7 D17
      OR=     K8 D17
      ANB
      MPS
      AND     M77  ; Don't temporarily use
      MOV     K0 D17
      MPP
      AND     M77  ; Don't temporarily use
      RST     L2079  ; Power Failure Door Open_PC
823   END
END_PROGRAM
